// TIA Portal V20 export
DATA_BLOCK "DB_PLC"   // DB7
// PLC-specific system data (C-305). Simulation is force-reset FALSE at every startup (OB100, C-305/C-403) regardless of retentivity - simulation mode must never survive a power cycle; start values only apply at download, not restart.
   VAR RETAIN
      Simulation : Bool := FALSE;
   END_VAR
BEGIN
END_DATA_BLOCK
